// SIMATIC S7-200 project (STEP 7-Micro/WIN), CPU 224 CN REL 02.01

SYMBOL_TABLE 辅助
QDF              M1.0     // l运转启动
ZBF              M1.1     // 转速交变试验
WBF              M1.2     // 温度交变试验
GBF              M1.3     // 干温交变试验
ZBJSFW           M1.4     // 转速交变计数复位
WBJSFW           M1.5     // 温度交变计数复位
GBJSFW           M1.6     // 干湿交变计数复位
ZBWQ             M1.7     // 转速交变温控启动
WBWQ             M2.0     // 温度交变温控启动
GBWQ             M2.1     // 干温交变温控启动
                 M2.2     // 1号加热
                 M2.3     // 2号加热
                 M2.4     // 3号加热
                 M2.5     // 4号加热
                 M2.6     // 5号加热
                 M2.7     // 加热启动
F1               M3.0     // 1号气阀开
F2               M3.1     // 2号气阀开
F3               M3.2     // 3号气阀开
F4               M3.3     // 4号气阀开
F5               M3.4     // 5号气阀开
ZFF              M3.5     // 进口总气阀开
PF1              M3.6     // 室温自控
PF2              M3.7     // 强制排风
PF3              M4.0     // 排风辅助
FGDW             M4.1     // 阀门开到位
FKDW             M4.2     // 阀门关到位
F55              M4.3     // 5号气阀开
FXF              M4.4     // 皮带放松辅助
LJF              M4.5     // 皮带拉紧辅助
FXXWF            M4.6     // 放松限位辅助
LJXWF            M4.7     // 皮带限位辅助
DILJF            M5.0     // 手控拉紧辅助
DIFXF            M5.1     // 手控放松辅助
DILJFF           M5.2     // 手控拉紧辅助1
DIFXFF           M5.3     // 手控放松辅助1
HBF              M5.4     // 恒速试验
JS1F             M6.0     // 1号进水辅助
JS2F             M6.1     // 2号进水辅助
JS3F             M6.2     // 3号进水辅助
JS4F             M6.3     // 4号进水辅助
JS5F             M6.4     // 5号进水辅助
PS1F             M6.5     // 1号排水辅助
PS2F             M6.6     // 2号排水辅助
PS3F             M6.7     // 3号排水辅助
PS4F             M7.0     // 4号排水辅助
PS5F             M7.1     // 5号排水辅助
PSF              M7.2     // 排水辅助
JSF              M7.3     // 进水辅助
YWSF             M7.4     // 总水箱上限辅助
YWXF             M7.5     // 总水箱下限辅助
FZ1              M7.6     // 液位控制辅助1
FZ2              M7.7     // 液位控制辅助2
FZ3              M8.0     // 液位控制辅助3
FZ4              M8.1     // 液位控制辅助4
YWXF1            M8.2     // 液位下限辅助1
YWXF2            M8.3     // 液位下限辅助2
YWXF3            M8.4     // 液位下限辅助3
YWXF4            M8.5     // 液位下限辅助4
YWXF5            M8.6     // 液位下限辅助5
CYF              M8.7     // 采样辅助
WCF              M9.0     // 试验完成
SSJS             T101     // 转速上升时间
HSJS             T102     // 转速恒速时间
JSJS             T103     // 转速下降时间
GSSJS            T104     // 干湿交变加水时间
GSSJG            T105     // 干湿交变无水时间
                 T106     // 温度交变时间1
                 T107     // 温度交变时间2
                 T108     // 温度交变时间3
                 T109     // 温度交变时间4
                 T110     // 温度交变时间5
JR1SK            T111     // 1号箱加热控制时间
JR2SK            T112     // 2号箱加热控制时间
JR3SK            T113     // 3号箱加热控制时间
JR4SK            T114     // 4号箱加热控制时间
JR5SK            T115     // 5号箱加热控制时间
JRSZK            T116     // 加热间隔2秒延时
JRSZKF           T117     // 加热间隔2秒延时辅助
                 T46      // 采样时间
END_SYMBOL_TABLE

SYMBOL_TABLE 输入
                 I0.0     // 转速
FK               I0.1     // 电阀到位
YW1S             I0.2     // 1号箱水位上限
YW1X             I0.3     // 1号箱水位下限
YW2S             I0.4     // 2号箱水位上限
YW2X             I0.5     // 2号箱水位下限
YW3S             I0.6     // 3号箱水位上限
YW3X             I0.7     // 3号箱水位下限
YW4S             I1.0     // 4号箱水位上限
YW4X             I1.1     // 4号箱水位下限
YW5S             I1.2     // 5号箱水位上限
YW5X             I1.3     // 5号箱水位下限
YWS              I1.4     // 总箱水位上限
YWX              I1.5     // 总箱水位下限
FXW              I2.0     // 放松限位
LJW              I2.1     // 拉紧限位
DILJXC           I2.2     // 手控皮带拉紧
DIFXXC           I2.3     // 手控皮带放松
QD               I2.4     // 试验启动
TZ               I2.5     // 试验停止
DIDFK            I2.6     // 电阀开
DIDFG            I2.7     // 电阀关
DILJ             I3.0     // 手控皮带拉紧
DIFX             I3.1     // 手控皮带放松
DYQD             I3.2     // 电源启动
DYTZ             I3.3     // 电源停止
XL               I3.4     // 泄漏
CS               I3.5     // 水泵出水管有水
END_SYMBOL_TABLE

SYMBOL_TABLE 输出
DY               Q0.0     // 总电源
JRK              Q0.1     // 加热控制
JR1              Q0.2     // 加热1号箱
JR2              Q0.3     // 加热2号箱
JR3              Q0.4     // 加热3号箱
JR4              Q0.5     // 加热4号箱
JR5              Q0.6     // 加热5号箱
DFK              Q0.7     // 电阀开
DFG              Q1.0     // 电阀关
LJ               Q1.1     // 电机拉紧
FX               Q2.0     // 电机放松
PF               Q2.1     // 排风扇
ZYF              Q2.2     // 增压阀F18
PYF              Q2.3     // 排空阀F19
QF1              Q2.4     // 1号箱气阀F12
QF2              Q2.5     // 2号箱气阀F13
QF3              Q2.6     // 3号箱气阀F14
QF4              Q2.7     // 4号箱气阀F15
QF5              Q3.0     // 5号箱气阀F16
ZQF              Q3.1     // 总控气阀FF17
JS1              Q3.2     // 1号箱进水F3
JS2              Q3.3     // 2号箱进水F4
JS3              Q3.4     // 3号箱进水F5
JS4              Q3.5     // 4号箱进水F6
JS5              Q3.6     // 5号箱进水F7
ZJS              Q3.7     // 总进水F1
ZPS              Q4.0     // 总排水F2
ZKF              Q4.1     // 总水箱控制F8
CKJQF            Q4.2     // 水泵出水管进气F11
JKPSF            Q4.3     // 水泵进水管排水F9
ZSXJY            Q4.4     // 总水箱加压(水盆回水)F10
NZ               Q4.5     // 逆转
SZ               Q4.6     // 顺转
END_SYMBOL_TABLE

SYMBOL_TABLE 变量
XTQD             VB201    // ＝0停止　＝1启动
ZDFX             VB202    // 转动方向＝0顺时运转　＝0逆时运转
SYLX             VB203    // 系统停止＝0　转速交变＝1　温度交变＝2　干交变＝3
PKQD             VB204    // 压力控制=0停止=1自动
YZZT             VB205    // 运转状态＝0停止＝1升速　＝2恒速　＝3降速
WKQD             VB206    // =0加热停止 =1加热启动
HKZ              VB207    // 扬程控制=0手控 =1自控
YWKZ             VB208    // 液位控制=0手控 =1自控
WBSL             VB209    // 温变数量
WBBK             VB210    // 温变步控
LLKZ             VB211    // 拉力控制=0停止=1自动
SBZT             VB212    // 试验状态=0正常 =1 泄漏 =2结束
XLCY             VB214    // 允许泄漏报警
ZPC              VD150    // 转速交变频次
WPC              VD154    // 温度交变频次
GPC              VD158    // 干湿交变频次
H                VW100    // 扬程
P                VW102    // 水箱压力
LL               VW104    // 皮带拉力
WD1              VW106    // 水温1
WD2              VW108    // 水温2
WD3              VW110    // 水温3
WD4              VW112    // 水温4
WD5              VW114    // 水温5
SW               VW116    // 室温
N                VW118    // 转速
FW               VW120    // 阀位
LLSD             VW122    // 拉力设定
PSD              VW124    // 压力设定
HSD              VW126    // 扬程设定
ZSJ              VW128    // 状态运行时间
WD1SD            VW130    // 温度设定1
WD2SD            VW132    // 温度设定2
WD3SD            VW134    // 温度设定3
WD4SD            VW136    // 温度设定4
WD5SD            VW138    // 温度设定5
SJSD1            VW140    // 时间设定1
SJSD2            VW142    // 时间设定2
SJSD3            VW144    // 时间设定3
SJSD4            VW146    // 时间设定4
SJSD5            VW148    // 时间设定5
WD1WC            VW306    // 1号箱温差
WD2WC            VW308    // 2号箱温差
WD3WC            VW310    // 3号箱温差
WD4WC            VW312    // 4号箱温差
WD5WC            VW314    // 5号箱温差
HMAX             VW316    // 扬程上限N
HMIN             VW318    // 扬程下限N
LLMAX            VW320    // 拉力上限N
LLMIN            VW322    // 拉力下限N
PMAX             VW356    // 压力上限
PMIN             VW358    // 压力下限
WD1WCF           VW378    // 1号箱温度差
WD2WCF           VW380    // 2号箱温度差
WD3WCF           VW382    // 3号箱温度差
WD4WCF           VW384    // 4号箱温度差
WD5WCF           VW386    // 5号箱温度差
END_SYMBOL_TABLE

ORGANIZATION_BLOCK 程序块:OB1
TITLE=程序注释
BEGIN
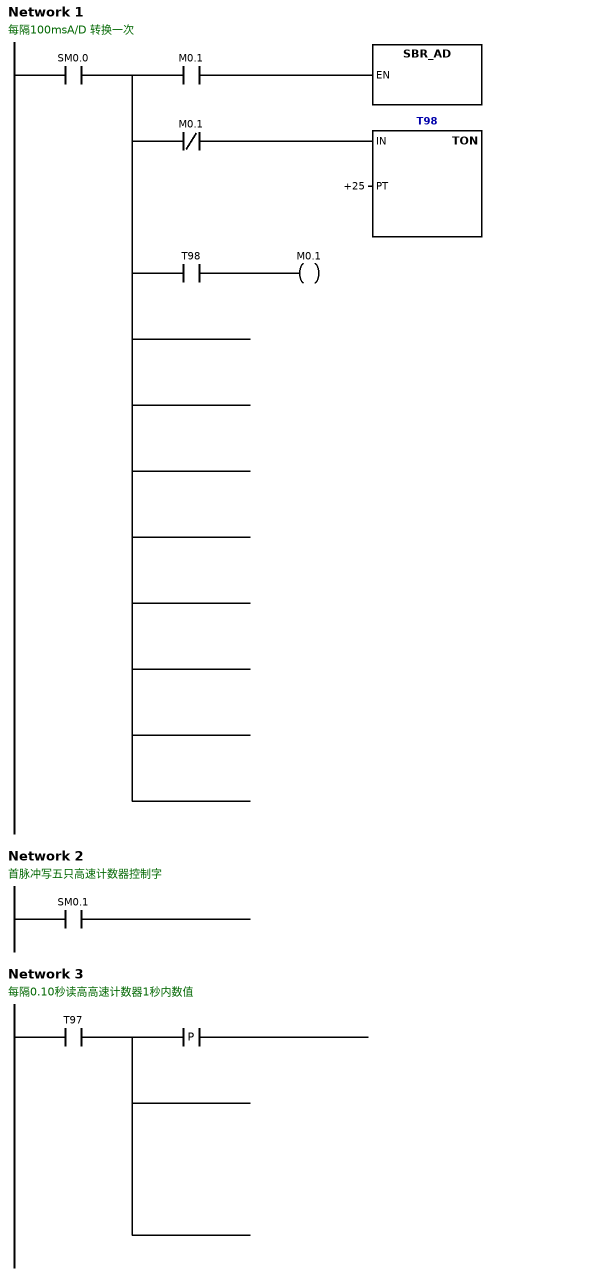
Network 1
// 每隔100msA/D 转换一次
// (network saved uncompiled; LAD cells follow)
// row 0: c0 -| |- SM0.0 v  c1 -| |- M0.1  c2 --  c3 [SBR_AD EN:=power@row0]
// row 1: c0 ^v  c1 -|/|- M0.1  c2 --  c3 [TON T98 IN:=power@row1, PT:=+25]
// row 2: c0 ^v  c3 [box]
// row 3: c0 ^v  c1 -| |- T98  c2 -( ) M0.1
// row 4: c0 ^v  c1 --
// row 5: c0 ^v  c1 --
// row 6: c0 ^v  c1 --
// row 7: c0 ^v  c1 --
// row 8: c0 ^v  c1 --
// row 9: c0 ^v  c1 --
// row 10: c0 ^v  c1 --
// row 11: c0 ^  c1 --
Network 2
// 首脉冲写五只高速计数器控制字
// (network saved uncompiled; LAD cells follow)
// row 0: c0 -| |- SM0.1  c1 --
Network 3
// 每隔0.10秒读高高速计数器1秒内数值
// (network saved uncompiled; LAD cells follow)
// row 0: c0 -| |- T97 v  c1 -|P|-  c2 --
// row 1: c0 ^v  c1 --
// row 2: c0 ^v
// row 3: c0 ^  c1 --
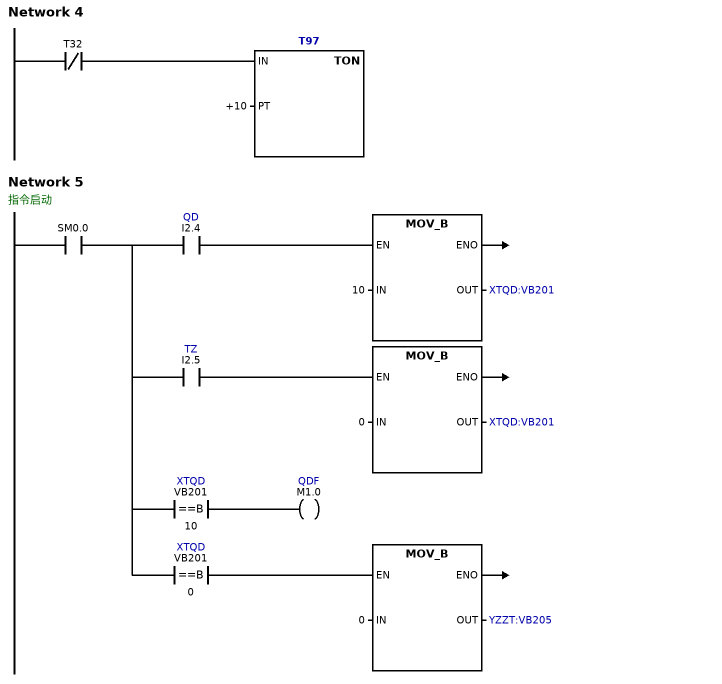
Network 4
LDN    T32
TON    T97, +10
Network 5
// 指令启动
LD     SM0.0
LPS
A      QD:I2.4
MOVB   10, XTQD:VB201
LRD
A      TZ:I2.5
MOVB   0, XTQD:VB201
LRD
AB=    XTQD:VB201, 10
=      QDF:M1.0
LPP
AB=    XTQD:VB201, 0
MOVB   0, YZZT:VB205
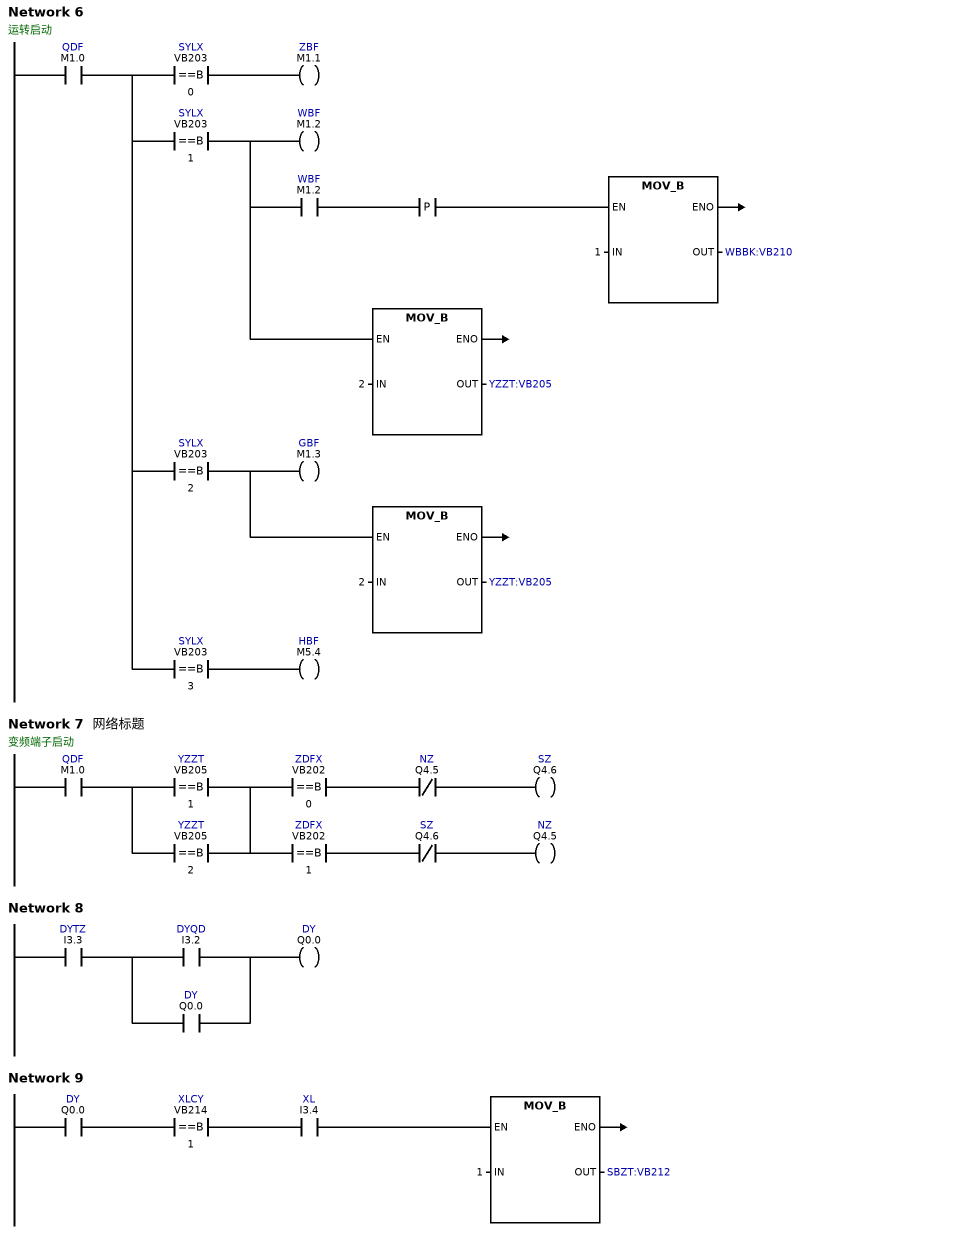
Network 6
// 运转启动
LD     QDF:M1.0
LPS
AB=    SYLX:VB203, 0
=      ZBF:M1.1
LRD
AB=    SYLX:VB203, 1
LPS
=      WBF:M1.2
A      WBF:M1.2
EU
MOVB   1, WBBK:VB210
LPP
MOVB   2, YZZT:VB205
LRD
AB=    SYLX:VB203, 2
=      GBF:M1.3
MOVB   2, YZZT:VB205
LPP
AB=    SYLX:VB203, 3
=      HBF:M5.4
Network 7 // 网络标题
// 变频端子启动
LD     QDF:M1.0
LDB=   YZZT:VB205, 1
OB=    YZZT:VB205, 2
ALD
LPS
AB=    ZDFX:VB202, 0
AN     NZ:Q4.5
=      SZ:Q4.6
LPP
AB=    ZDFX:VB202, 1
AN     SZ:Q4.6
=      NZ:Q4.5
Network 8
LD     DYTZ:I3.3
LD     DYQD:I3.2
O      DY:Q0.0
ALD
=      DY:Q0.0
Network 9
LD     DY:Q0.0
AB=    XLCY:VB214, 1
A      XL:I3.4
MOVB   1, SBZT:VB212
Network 18 // 网络标题
// 网络注释
END_ORGANIZATION_BLOCK

SUBROUTINE_BLOCK SBR_AD:SBR0
TITLE=子例行程序注释
BEGIN
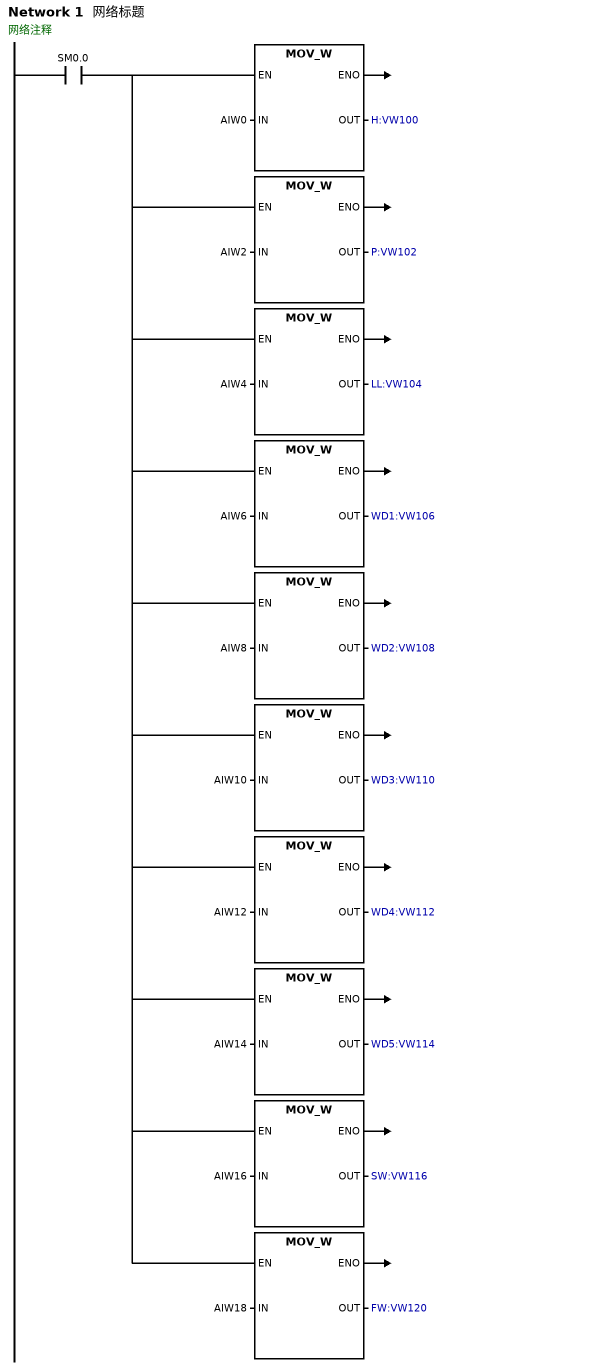
Network 1 // 网络标题
// 网络注释
LD     SM0.0
MOVW   AIW0, H:VW100
MOVW   AIW2, P:VW102
MOVW   AIW4, LL:VW104
MOVW   AIW6, WD1:VW106
MOVW   AIW8, WD2:VW108
MOVW   AIW10, WD3:VW110
MOVW   AIW12, WD4:VW112
MOVW   AIW14, WD5:VW114
MOVW   AIW16, SW:VW116
MOVW   AIW18, FW:VW120
Network 11 // 网络标题
// 网络注释
END_SUBROUTINE_BLOCK

SUBROUTINE_BLOCK 干湿交变:SBR1
TITLE=子例行程序注释
BEGIN
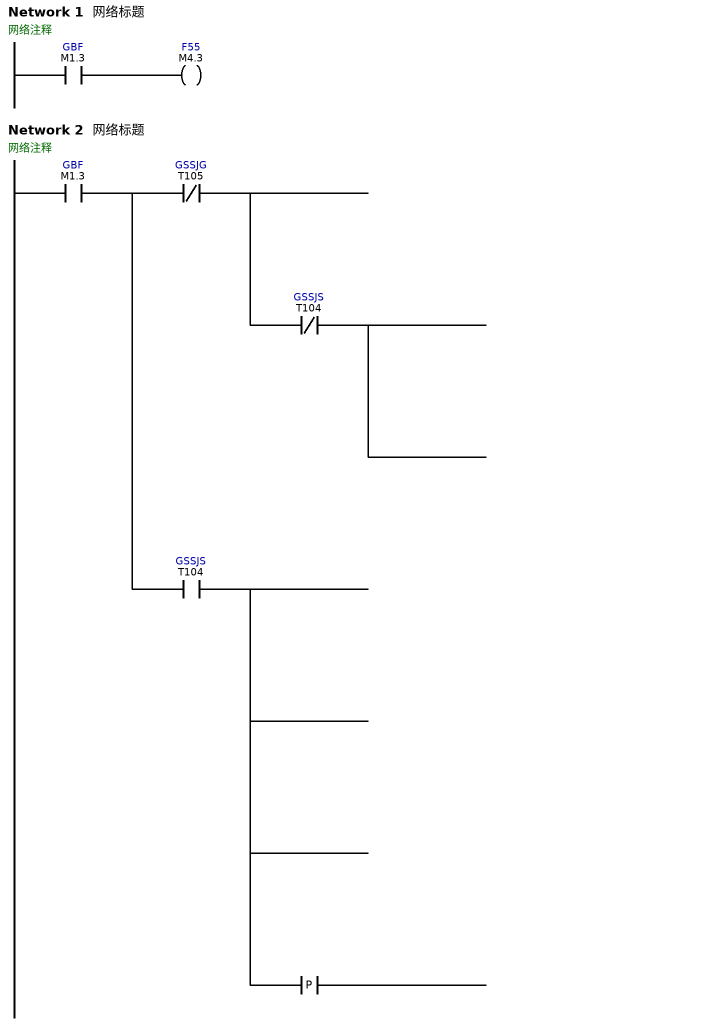
Network 1 // 网络标题
// 网络注释
LD     GBF:M1.3
=      F55:M4.3
Network 2 // 网络标题
// 网络注释
// (network saved uncompiled; LAD cells follow)
// row 0: c0 -| |- GBF:M1.3 v  c1 -|/|- GSSJG:T105 v  c2 --
// row 1: c0 ^v  c1 ^v
// row 2: c0 ^v  c1 ^  c2 -|/|- GSSJS:T104 v  c3 --
// row 3: c0 ^v  c2 ^v
// row 4: c0 ^v  c2 ^  c3 --
// row 5: c0 ^v
// row 6: c0 ^  c1 -| |- GSSJS:T104 v  c2 --
// row 7: c1 ^v
// row 8: c1 ^v  c2 --
// row 9: c1 ^v
// row 10: c1 ^v  c2 --
// row 11: c1 ^v
// row 12: c1 ^  c2 -|P|-  c3 --
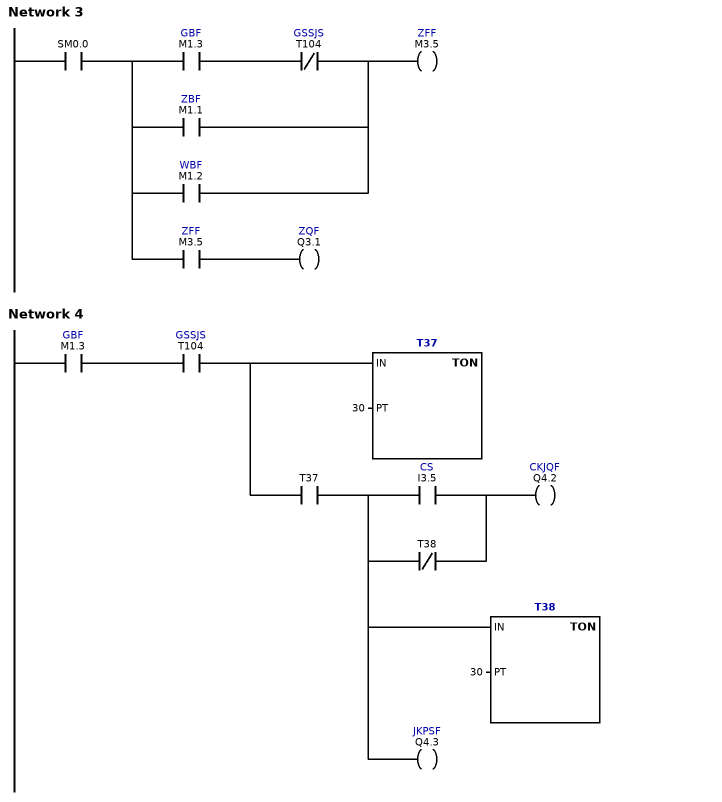
Network 3
LD     SM0.0
LPS
LD     GBF:M1.3
AN     GSSJS:T104
O      ZBF:M1.1
O      WBF:M1.2
ALD
=      ZFF:M3.5
LPP
A      ZFF:M3.5
=      ZQF:Q3.1
Network 4
LD     GBF:M1.3
A      GSSJS:T104
TON    T37, 30
A      T37
LPS
LD     CS:I3.5
ON     T38
ALD
=      CKJQF:Q4.2
LPP
TON    T38, 30
=      JKPSF:Q4.3
END_SUBROUTINE_BLOCK

SUBROUTINE_BLOCK 水温控制:SBR2
TITLE=子例行程序注释
BEGIN
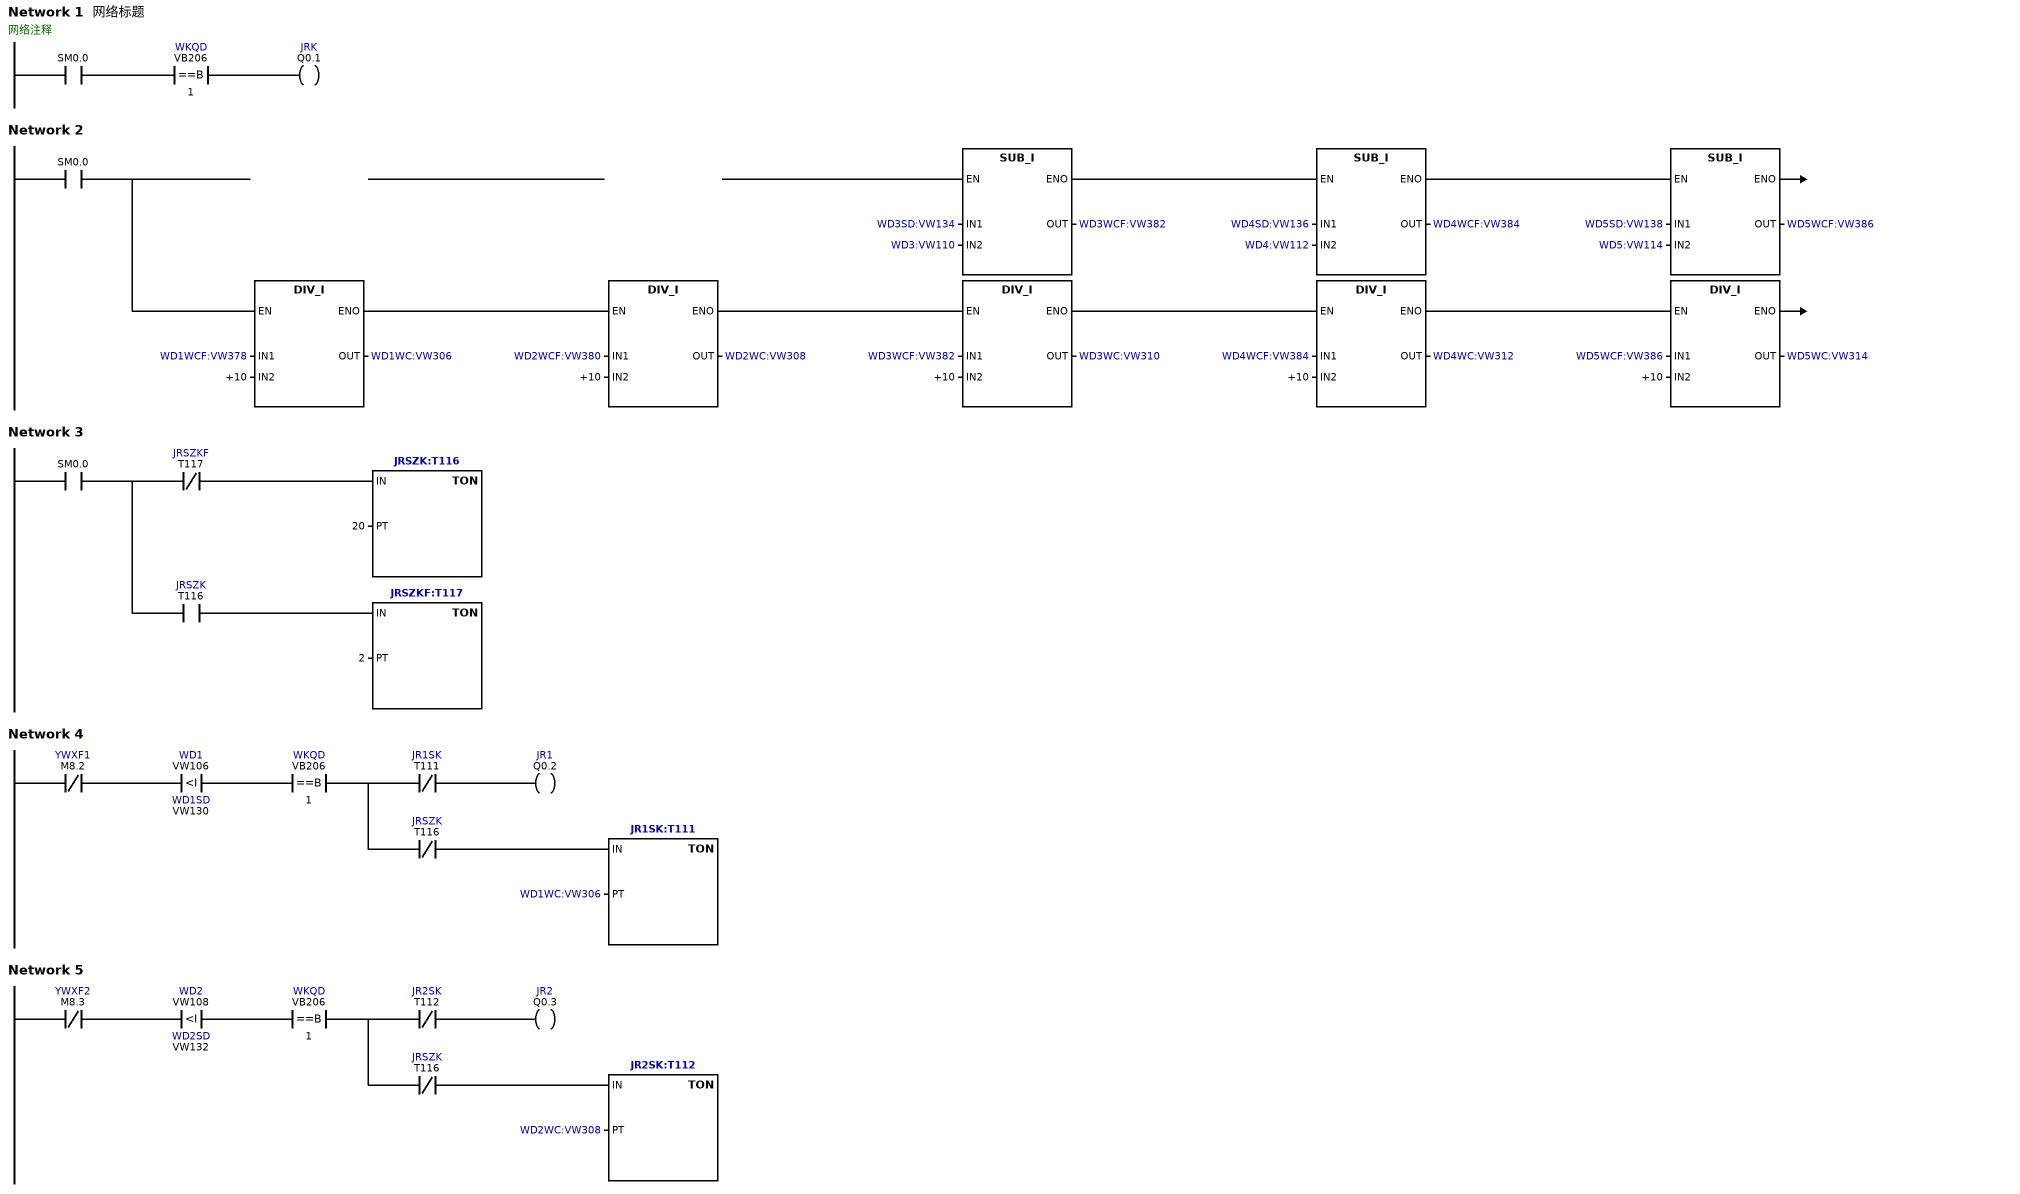
Network 1 // 网络标题
// 网络注释
LD     SM0.0
AB=    WKQD:VB206, 1
=      JRK:Q0.1
Network 2
// (network saved uncompiled; LAD cells follow)
// row 0: c0 -| |- SM0.0 v  c1 --  c3 --  c4 --  c6 --  c7 --  c8 [SUB_I EN:=power@row0, IN1:=WD3SD:VW134, IN2:=WD3:VW110, ENO=>power, OUT=>WD3WCF:VW382]  c9 --  c10 --  c11 [SUB_I EN:=power@row0, IN1:=WD4SD:VW136, IN2:=WD4:VW112, ENO=>power, OUT=>WD4WCF:VW384]  c12 --  c13 --  c14 [SUB_I EN:=power@row0, IN1:=WD5SD:VW138, IN2:=WD5:VW114, ENO=>power, OUT=>WD5WCF:VW386]  c15 ->
// row 1: c0 ^v  c8 [box]  c11 [box]  c14 [box]
// row 2: c0 ^  c1 --  c2 [DIV_I EN:=power@row2, IN1:=WD1WCF:VW378, IN2:=+10, ENO=>power, OUT=>WD1WC:VW306]  c3 --  c4 --  c5 [DIV_I EN:=power@row2, IN1:=WD2WCF:VW380, IN2:=+10, ENO=>power, OUT=>WD2WC:VW308]  c6 --  c7 --  c8 [DIV_I EN:=power@row2, IN1:=WD3WCF:VW382, IN2:=+10, ENO=>power, OUT=>WD3WC:VW310]  c9 --  c10 --  c11 [DIV_I EN:=power@row2, IN1:=WD4WCF:VW384, IN2:=+10, ENO=>power, OUT=>WD4WC:VW312]  c12 --  c13 --  c14 [DIV_I EN:=power@row2, IN1:=WD5WCF:VW386, IN2:=+10, ENO=>power, OUT=>WD5WC:VW314]  c15 ->
// row 3: c2 [box]  c5 [box]  c8 [box]  c11 [box]  c14 [box]
Network 3
LD     SM0.0
LPS
AN     JRSZKF:T117
TON    JRSZK:T116, 20
LPP
A      JRSZK:T116
TON    JRSZKF:T117, 2
Network 4
LDN    YWXF1:M8.2
AW<    WD1:VW106, WD1SD:VW130
AB=    WKQD:VB206, 1
LPS
AN     JR1SK:T111
=      JR1:Q0.2
LPP
AN     JRSZK:T116
TON    JR1SK:T111, WD1WC:VW306
Network 5
LDN    YWXF2:M8.3
AW<    WD2:VW108, WD2SD:VW132
AB=    WKQD:VB206, 1
LPS
AN     JR2SK:T112
=      JR2:Q0.3
LPP
AN     JRSZK:T116
TON    JR2SK:T112, WD2WC:VW308
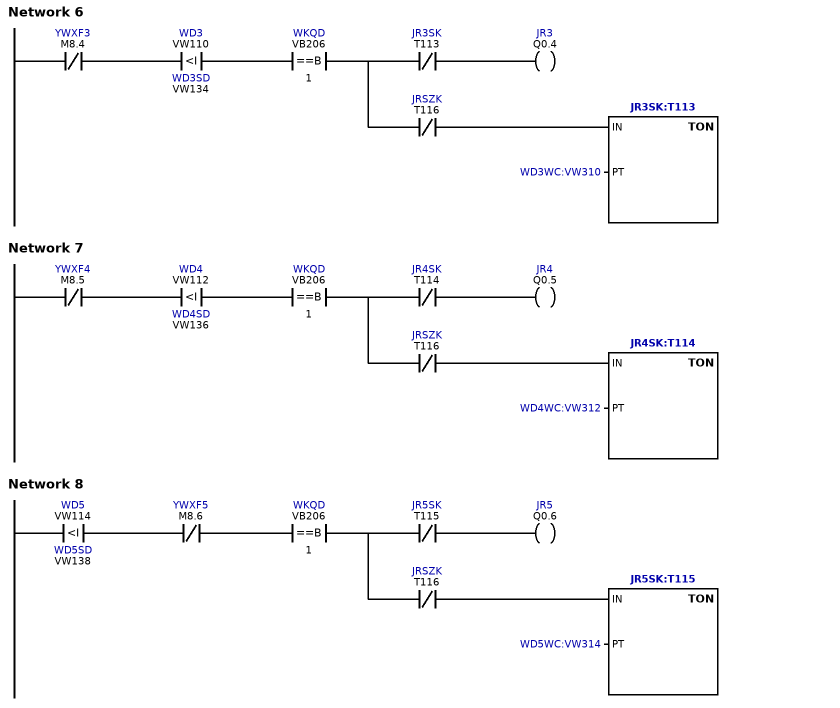
Network 6
LDN    YWXF3:M8.4
AW<    WD3:VW110, WD3SD:VW134
AB=    WKQD:VB206, 1
LPS
AN     JR3SK:T113
=      JR3:Q0.4
LPP
AN     JRSZK:T116
TON    JR3SK:T113, WD3WC:VW310
Network 7
LDN    YWXF4:M8.5
AW<    WD4:VW112, WD4SD:VW136
AB=    WKQD:VB206, 1
LPS
AN     JR4SK:T114
=      JR4:Q0.5
LPP
AN     JRSZK:T116
TON    JR4SK:T114, WD4WC:VW312
Network 8
LDW<   WD5:VW114, WD5SD:VW138
AN     YWXF5:M8.6
AB=    WKQD:VB206, 1
LPS
AN     JR5SK:T115
=      JR5:Q0.6
LPP
AN     JRSZK:T116
TON    JR5SK:T115, WD5WC:VW314
END_SUBROUTINE_BLOCK

SUBROUTINE_BLOCK 皮带拉力:SBR4
TITLE=子例行程序注释
BEGIN
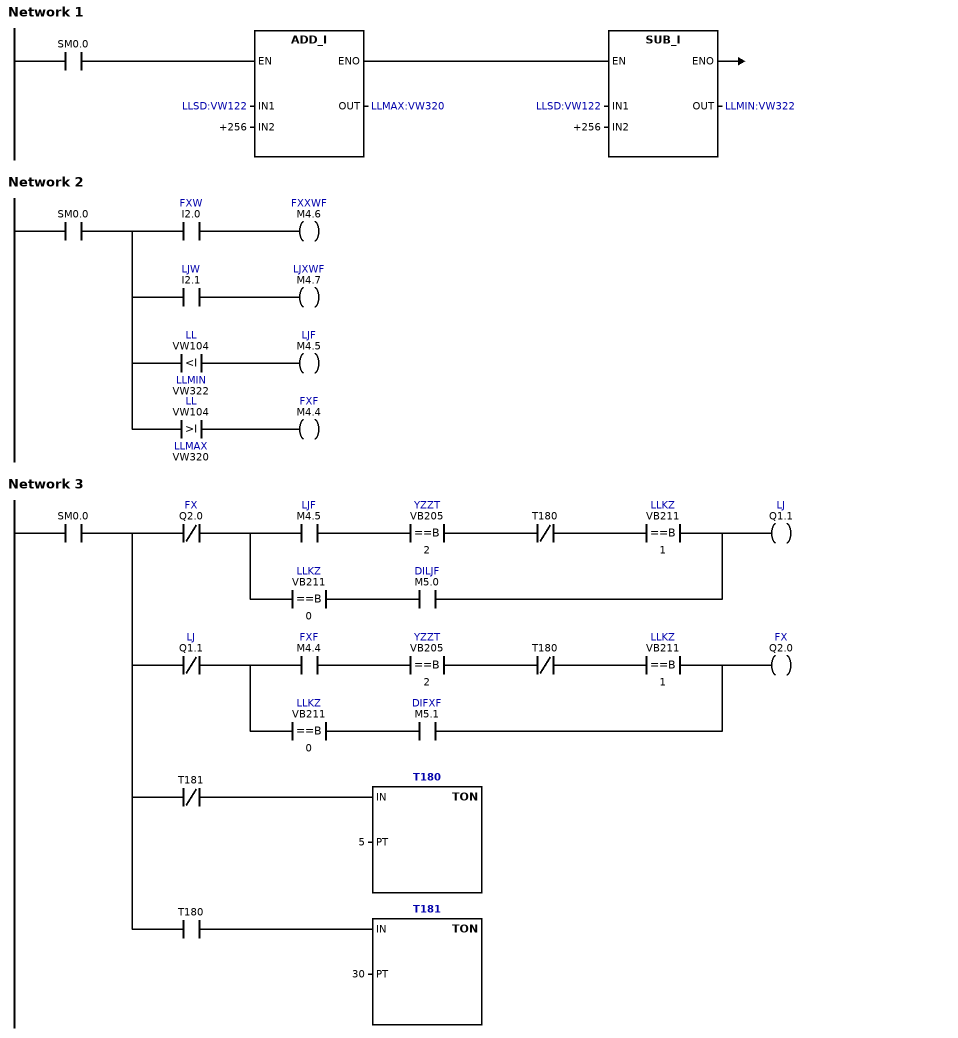
Network 1
LD     SM0.0
MOVW   LLSD:VW122, LLMAX:VW320
AENO
+I     +256, LLMAX:VW320
AENO
MOVW   LLSD:VW122, LLMIN:VW322
-I     +256, LLMIN:VW322
Network 2
LD     SM0.0
LPS
A      FXW:I2.0
=      FXXWF:M4.6
LRD
A      LJW:I2.1
=      LJXWF:M4.7
LRD
AW<    LL:VW104, LLMIN:VW322
=      LJF:M4.5
LPP
AW>    LL:VW104, LLMAX:VW320
=      FXF:M4.4
Network 3
LD     SM0.0
LPS
AN     FX:Q2.0
LD     LJF:M4.5
AB=    YZZT:VB205, 2
AN     T180
AB=    LLKZ:VB211, 1
LDB=   LLKZ:VB211, 0
A      DILJF:M5.0
OLD
ALD
=      LJ:Q1.1
LRD
AN     LJ:Q1.1
LD     FXF:M4.4
AB=    YZZT:VB205, 2
AN     T180
AB=    LLKZ:VB211, 1
LDB=   LLKZ:VB211, 0
A      DIFXF:M5.1
OLD
ALD
=      FX:Q2.0
LPP
LPS
AN     T181
TON    T180, 5
LPP
A      T180
TON    T181, 30
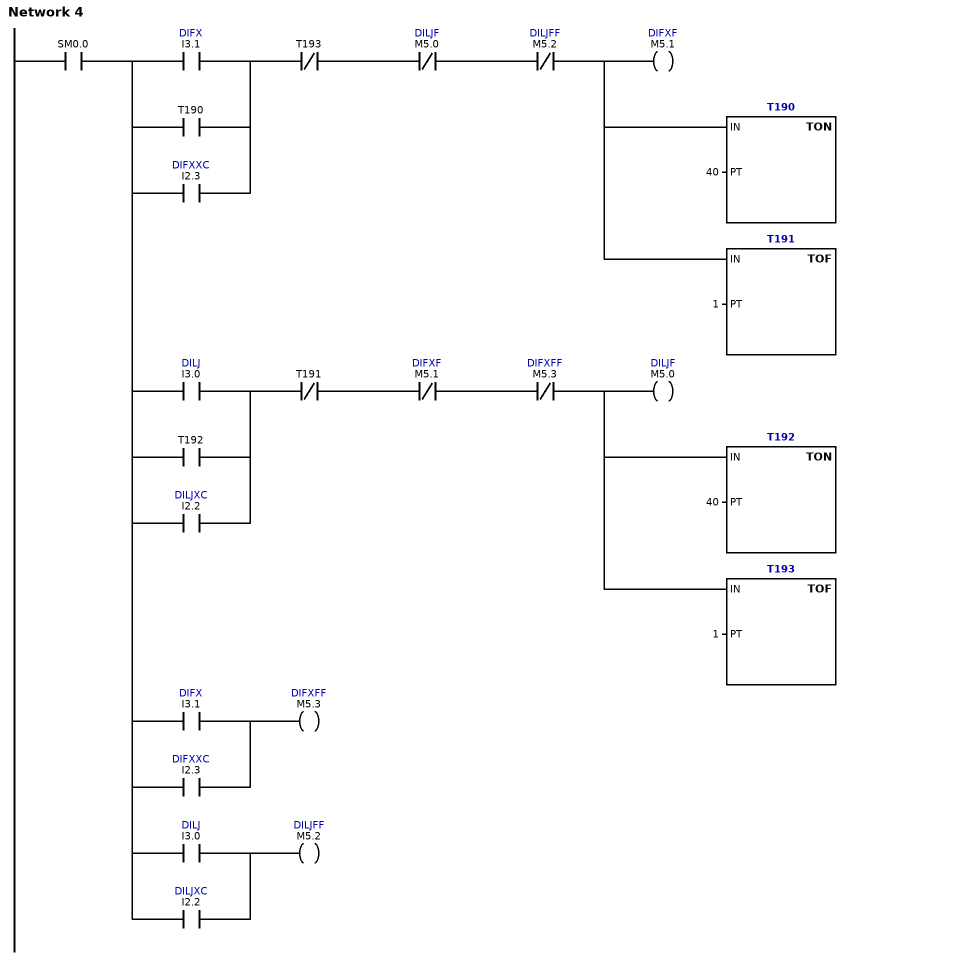
Network 4
LD     SM0.0
LPS
LD     DIFX:I3.1
O      T190
O      DIFXXC:I2.3
AN     T193
AN     DILJF:M5.0
AN     DILJFF:M5.2
ALD
=      DIFXF:M5.1
TON    T190, 40
TOF    T191, 1
LRD
LD     DILJ:I3.0
O      T192
O      DILJXC:I2.2
AN     T191
AN     DIFXF:M5.1
AN     DIFXFF:M5.3
ALD
=      DILJF:M5.0
TON    T192, 40
TOF    T193, 1
LRD
LD     DIFX:I3.1
O      DIFXXC:I2.3
ALD
=      DIFXFF:M5.3
LPP
LD     DILJ:I3.0
O      DILJXC:I2.2
ALD
=      DILJFF:M5.2
END_SUBROUTINE_BLOCK

SUBROUTINE_BLOCK HSC_清零:SBR5
TITLE=子例行程序注释
BEGIN
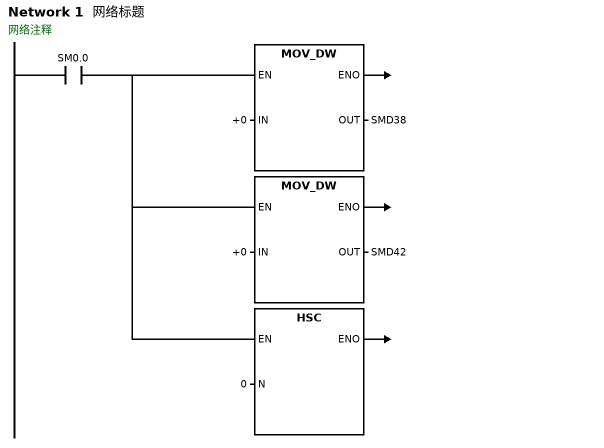
Network 1 // 网络标题
// 网络注释
LD     SM0.0
MOVD   +0, SMD38
MOVD   +0, SMD42
HSC    0
END_SUBROUTINE_BLOCK

SUBROUTINE_BLOCK 温度交变:SBR6
TITLE=子例行程序注释
BEGIN
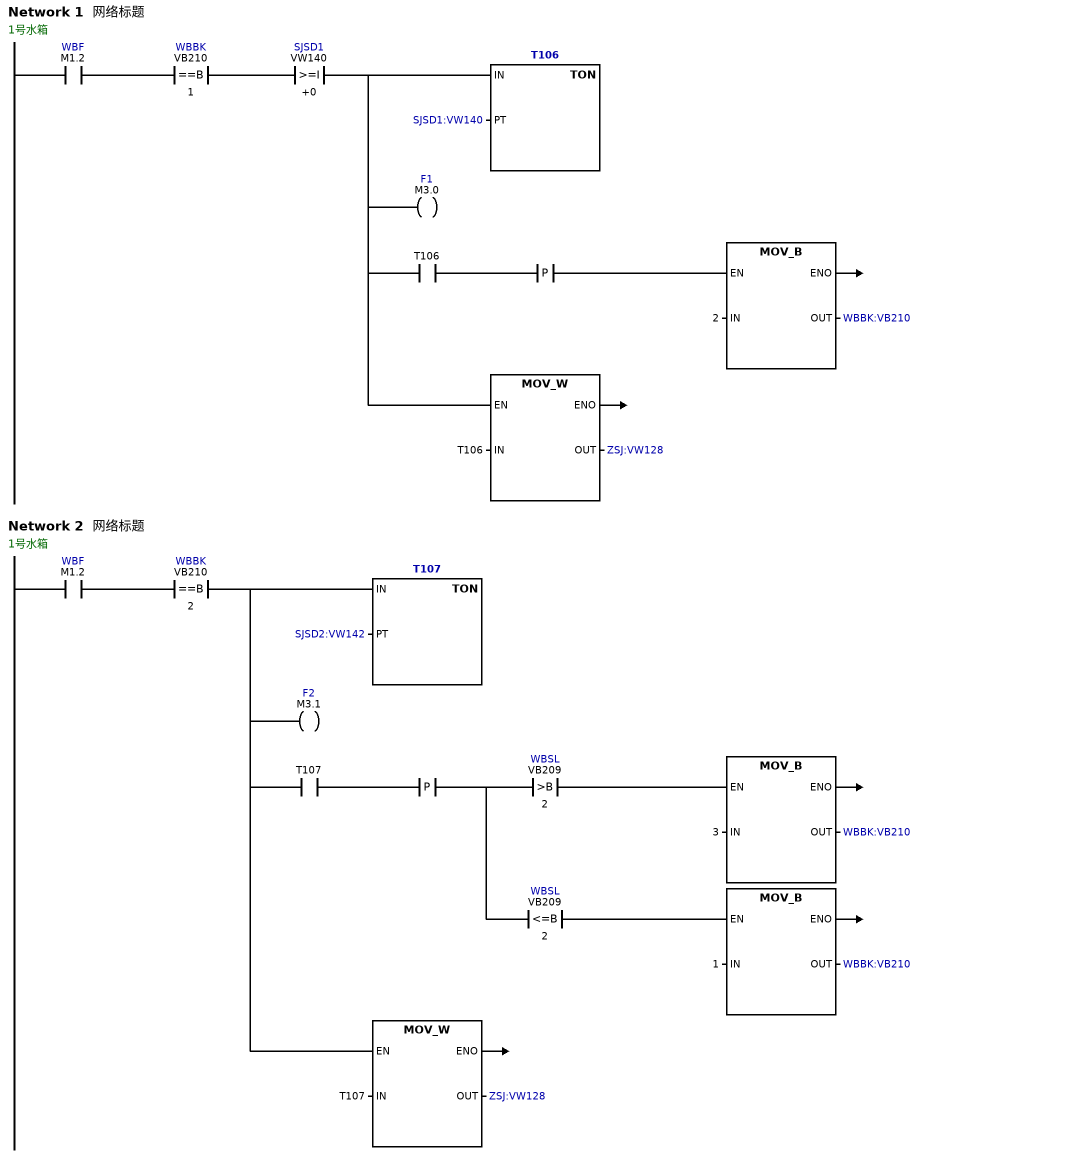
Network 1 // 网络标题
// 1号水箱
LD     WBF:M1.2
AB=    WBBK:VB210, 1
AW>=   SJSD1:VW140, +0
LPS
TON    T106, SJSD1:VW140
=      F1:M3.0
A      T106
EU
MOVB   2, WBBK:VB210
LPP
MOVW   T106, ZSJ:VW128
Network 2 // 网络标题
// 1号水箱
LD     WBF:M1.2
AB=    WBBK:VB210, 2
LPS
TON    T107, SJSD2:VW142
=      F2:M3.1
A      T107
EU
LPS
AB>    WBSL:VB209, 2
MOVB   3, WBBK:VB210
LPP
AB<=   WBSL:VB209, 2
MOVB   1, WBBK:VB210
LPP
MOVW   T107, ZSJ:VW128
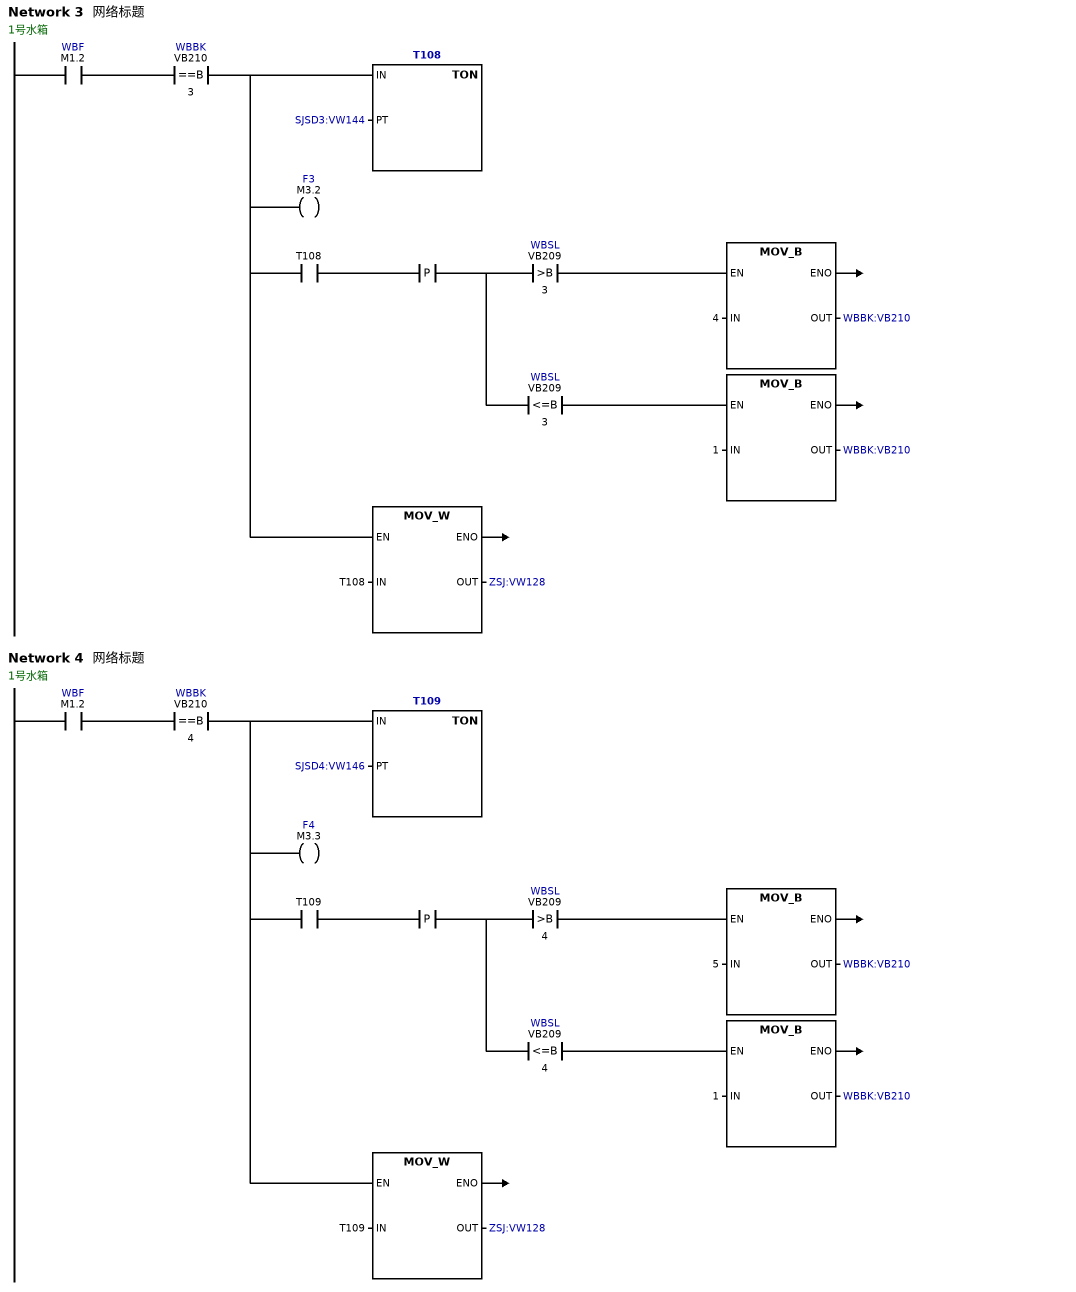
Network 3 // 网络标题
// 1号水箱
LD     WBF:M1.2
AB=    WBBK:VB210, 3
LPS
TON    T108, SJSD3:VW144
=      F3:M3.2
A      T108
EU
LPS
AB>    WBSL:VB209, 3
MOVB   4, WBBK:VB210
LPP
AB<=   WBSL:VB209, 3
MOVB   1, WBBK:VB210
LPP
MOVW   T108, ZSJ:VW128
Network 4 // 网络标题
// 1号水箱
LD     WBF:M1.2
AB=    WBBK:VB210, 4
LPS
TON    T109, SJSD4:VW146
=      F4:M3.3
A      T109
EU
LPS
AB>    WBSL:VB209, 4
MOVB   5, WBBK:VB210
LPP
AB<=   WBSL:VB209, 4
MOVB   1, WBBK:VB210
LPP
MOVW   T109, ZSJ:VW128
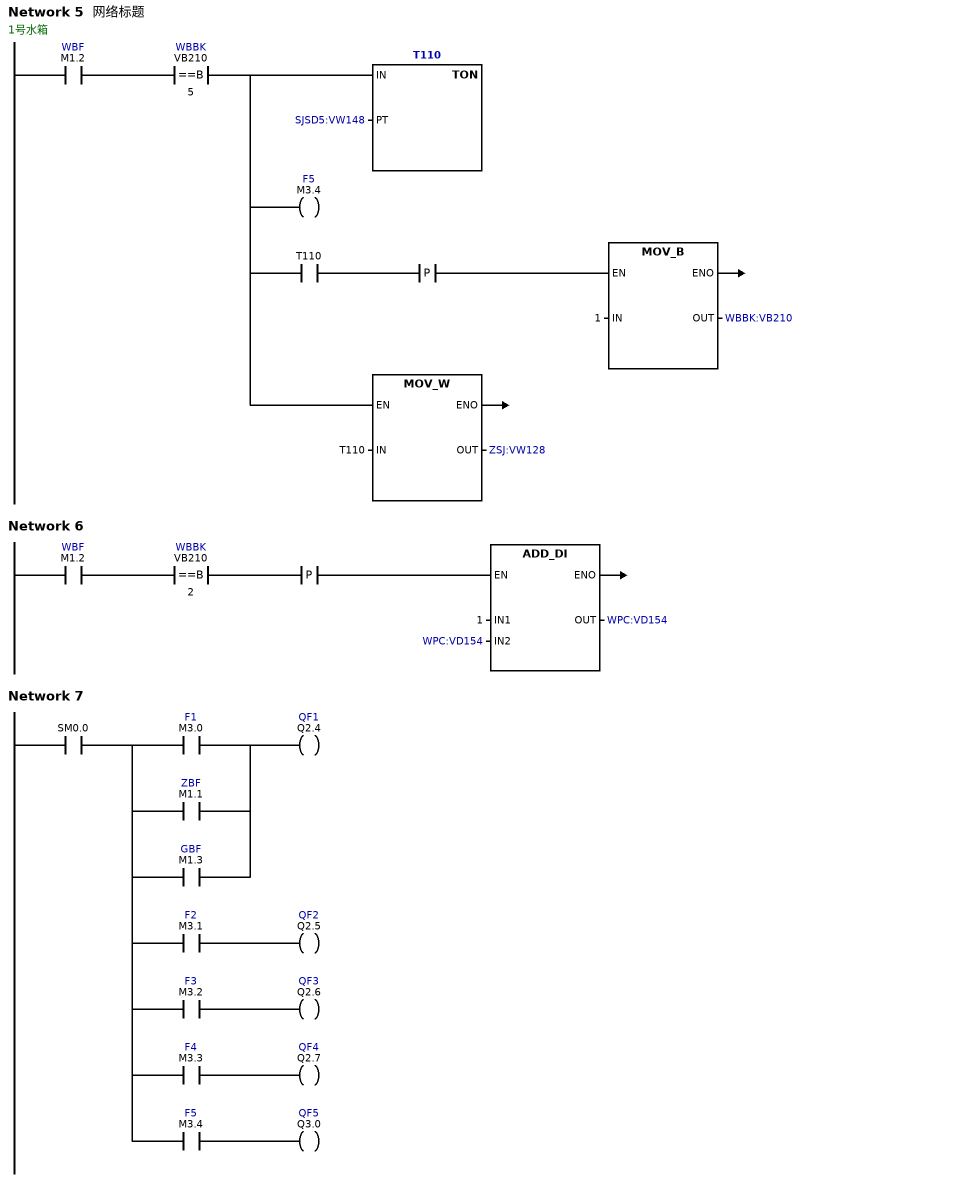
Network 5 // 网络标题
// 1号水箱
LD     WBF:M1.2
AB=    WBBK:VB210, 5
LPS
TON    T110, SJSD5:VW148
=      F5:M3.4
A      T110
EU
MOVB   1, WBBK:VB210
LPP
MOVW   T110, ZSJ:VW128
Network 6
LD     WBF:M1.2
AB=    WBBK:VB210, 2
EU
+D     1, WPC:VD154
Network 7
LD     SM0.0
LPS
LD     F1:M3.0
O      ZBF:M1.1
O      GBF:M1.3
ALD
=      QF1:Q2.4
LPP
LPS
A      F2:M3.1
=      QF2:Q2.5
LRD
A      F3:M3.2
=      QF3:Q2.6
LRD
A      F4:M3.3
=      QF4:Q2.7
LPP
A      F5:M3.4
=      QF5:Q3.0
END_SUBROUTINE_BLOCK

SUBROUTINE_BLOCK 液位控制:SBR7
TITLE=子程序注释
BEGIN
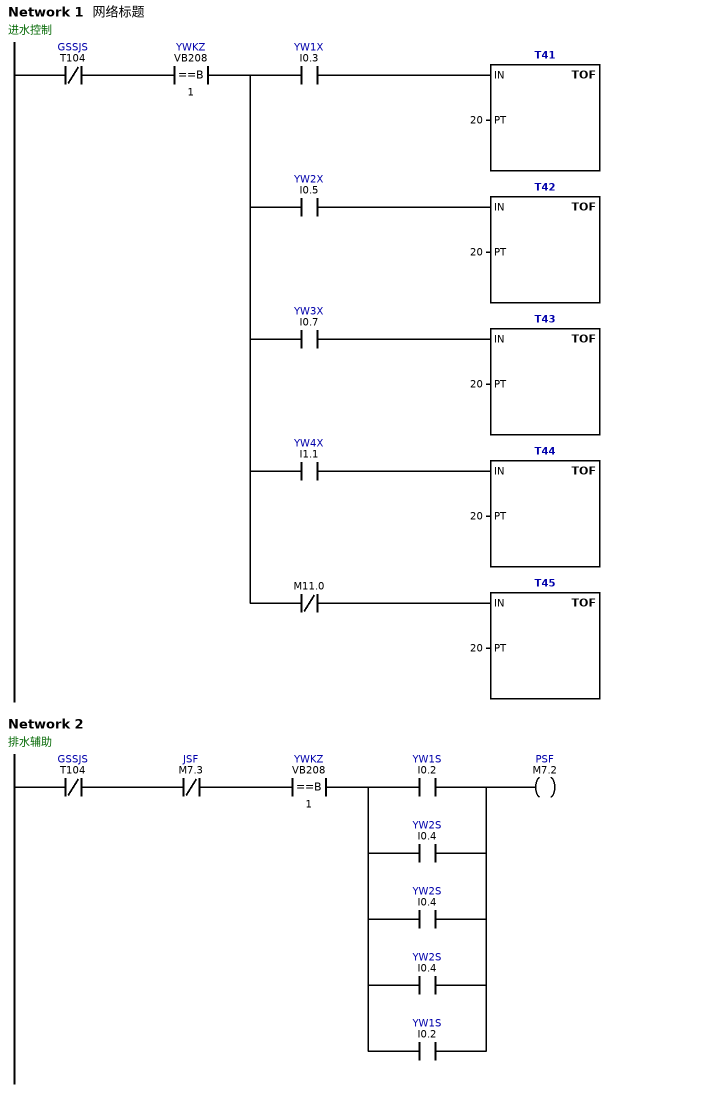
Network 1 // 网络标题
// 进水控制
LDN    GSSJS:T104
AB=    YWKZ:VB208, 1
LPS
A      YW1X:I0.3
TOF    T41, 20
LRD
A      YW2X:I0.5
TOF    T42, 20
LRD
A      YW3X:I0.7
TOF    T43, 20
LRD
A      YW4X:I1.1
TOF    T44, 20
LPP
AN     M11.0
TOF    T45, 20
Network 2
// 排水辅助
LDN    GSSJS:T104
AN     JSF:M7.3
AB=    YWKZ:VB208, 1
LD     YW1S:I0.2
O      YW2S:I0.4
O      YW2S:I0.4
O      YW2S:I0.4
O      YW1S:I0.2
ALD
=      PSF:M7.2
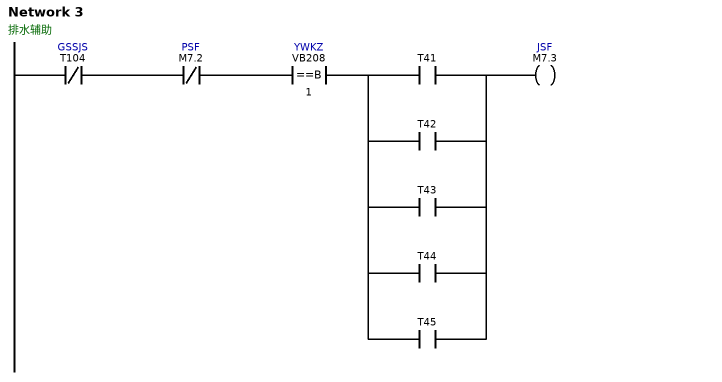
Network 3
// 排水辅助
LDN    GSSJS:T104
AN     PSF:M7.2
AB=    YWKZ:VB208, 1
LD     T41
O      T42
O      T43
O      T44
O      T45
ALD
=      JSF:M7.3
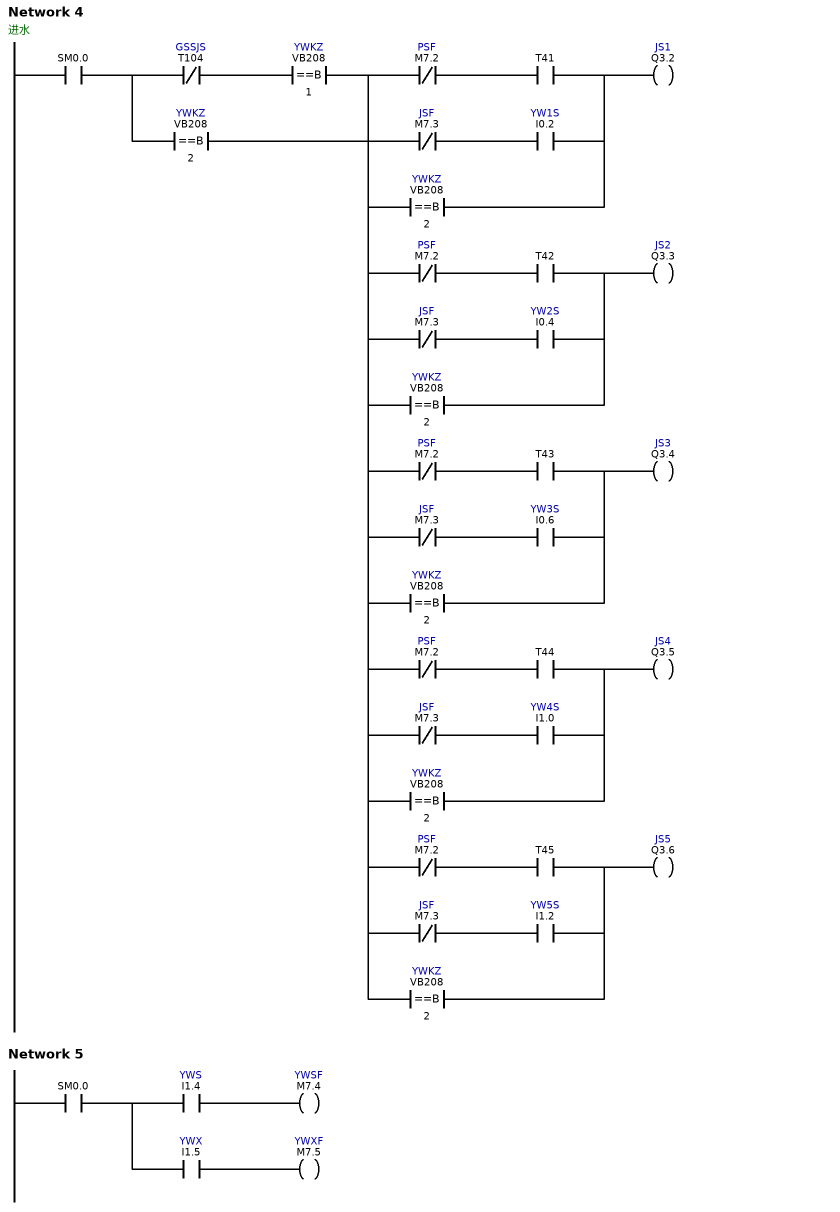
Network 4
// 进水
LD     SM0.0
LDN    GSSJS:T104
AB=    YWKZ:VB208, 1
OB=    YWKZ:VB208, 2
ALD
LPS
LDN    PSF:M7.2
A      T41
LDN    JSF:M7.3
A      YW1S:I0.2
OLD
OB=    YWKZ:VB208, 2
ALD
=      JS1:Q3.2
LRD
LDN    PSF:M7.2
A      T42
LDN    JSF:M7.3
A      YW2S:I0.4
OLD
OB=    YWKZ:VB208, 2
ALD
=      JS2:Q3.3
LRD
LDN    PSF:M7.2
A      T43
LDN    JSF:M7.3
A      YW3S:I0.6
OLD
OB=    YWKZ:VB208, 2
ALD
=      JS3:Q3.4
LRD
LDN    PSF:M7.2
A      T44
LDN    JSF:M7.3
A      YW4S:I1.0
OLD
OB=    YWKZ:VB208, 2
ALD
=      JS4:Q3.5
LPP
LDN    PSF:M7.2
A      T45
LDN    JSF:M7.3
A      YW5S:I1.2
OLD
OB=    YWKZ:VB208, 2
ALD
=      JS5:Q3.6
Network 5
LD     SM0.0
LPS
A      YWS:I1.4
=      YWSF:M7.4
LPP
A      YWX:I1.5
=      YWXF:M7.5
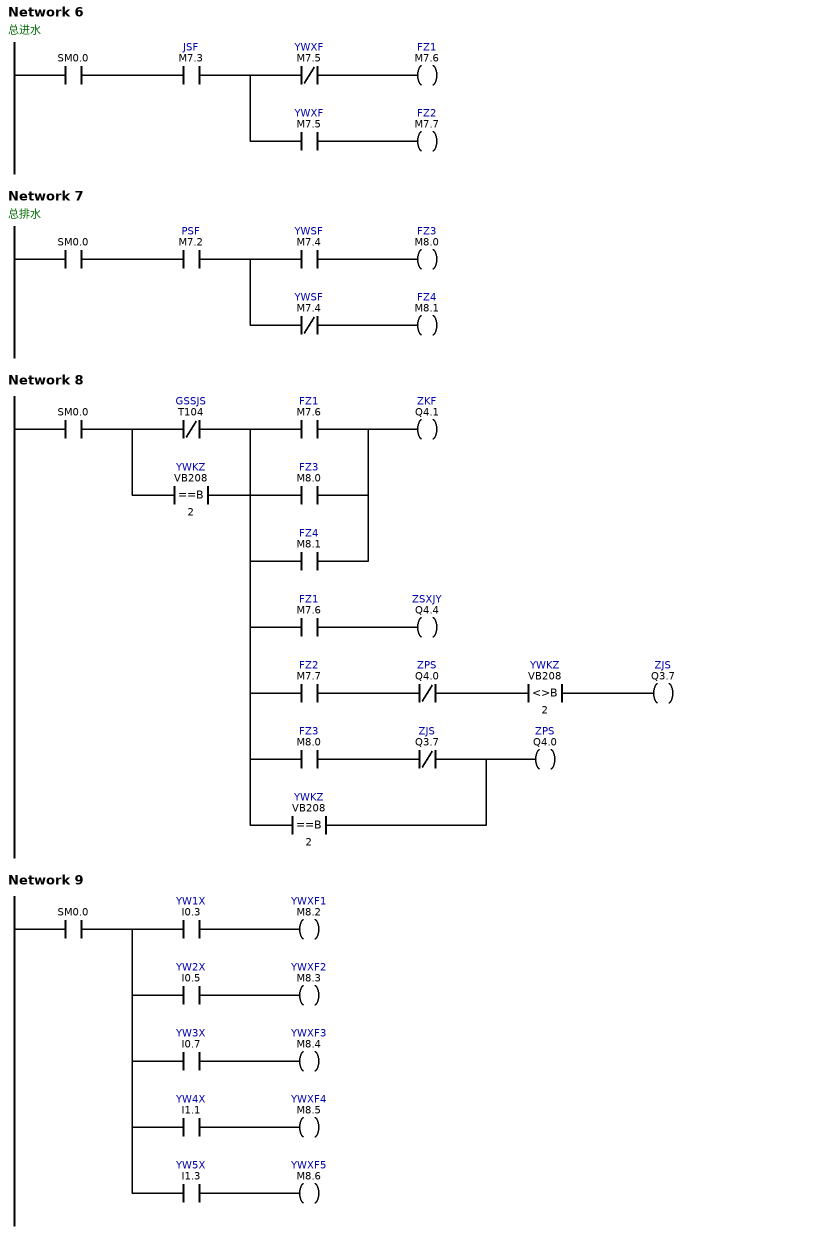
Network 6
// 总进水
LD     SM0.0
A      JSF:M7.3
LPS
AN     YWXF:M7.5
=      FZ1:M7.6
LPP
A      YWXF:M7.5
=      FZ2:M7.7
Network 7
// 总排水
LD     SM0.0
A      PSF:M7.2
LPS
A      YWSF:M7.4
=      FZ3:M8.0
LPP
AN     YWSF:M7.4
=      FZ4:M8.1
Network 8
LD     SM0.0
LDN    GSSJS:T104
OB=    YWKZ:VB208, 2
ALD
LPS
LD     FZ1:M7.6
O      FZ3:M8.0
O      FZ4:M8.1
ALD
=      ZKF:Q4.1
LRD
LPS
A      FZ1:M7.6
=      ZSXJY:Q4.4
LPP
A      FZ2:M7.7
AN     ZPS:Q4.0
AB<>   YWKZ:VB208, 2
=      ZJS:Q3.7
LPP
LD     FZ3:M8.0
AN     ZJS:Q3.7
OB=    YWKZ:VB208, 2
ALD
=      ZPS:Q4.0
Network 9
LD     SM0.0
LPS
A      YW1X:I0.3
=      YWXF1:M8.2
LRD
A      YW2X:I0.5
=      YWXF2:M8.3
LRD
A      YW3X:I0.7
=      YWXF3:M8.4
LRD
A      YW4X:I1.1
=      YWXF4:M8.5
LPP
A      YW5X:I1.3
=      YWXF5:M8.6
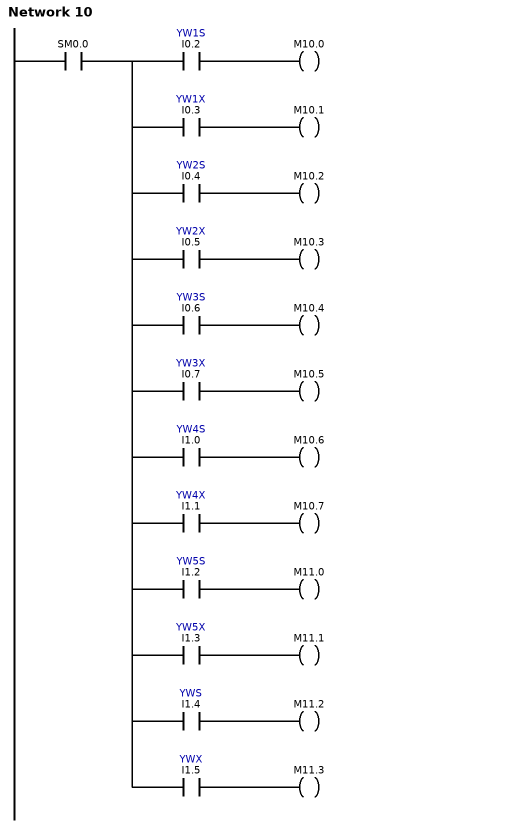
Network 10
LD     SM0.0
LPS
A      YW1S:I0.2
=      M10.0
LRD
A      YW1X:I0.3
=      M10.1
LRD
A      YW2S:I0.4
=      M10.2
LRD
A      YW2X:I0.5
=      M10.3
LRD
A      YW3S:I0.6
=      M10.4
LRD
A      YW3X:I0.7
=      M10.5
LRD
A      YW4S:I1.0
=      M10.6
LRD
A      YW4X:I1.1
=      M10.7
LRD
A      YW5S:I1.2
=      M11.0
LRD
A      YW5X:I1.3
=      M11.1
LRD
A      YWS:I1.4
=      M11.2
LPP
A      YWX:I1.5
=      M11.3
END_SUBROUTINE_BLOCK

SUBROUTINE_BLOCK HSC_初始化:SBR8
TITLE=子例行程序注释
BEGIN
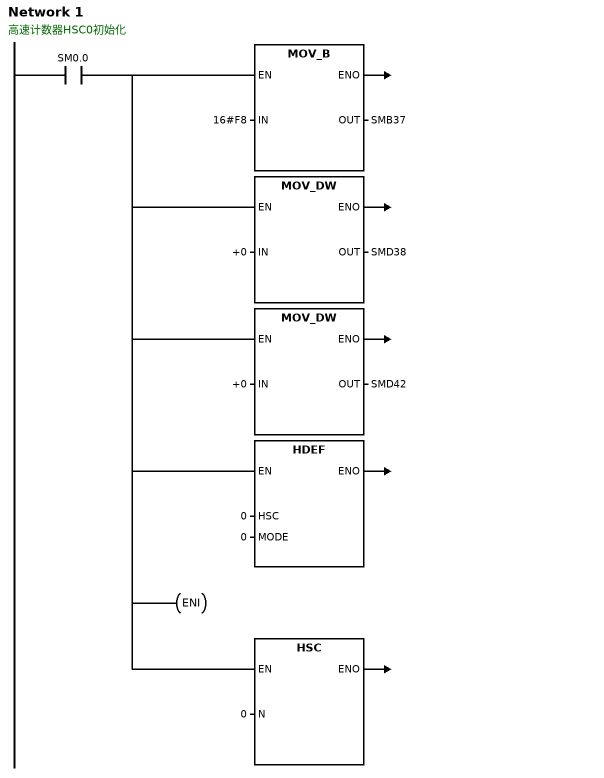
Network 1
// 高速计数器HSC0初始化
//设置控制位：向上计数；已启用；
//载入CV
//载入PV
LD     SM0.0
MOVB   16#F8, SMB37
MOVD   +0, SMD38
MOVD   +0, SMD42
HDEF   0, 0
ENI
HSC    0
Network 2 // 网络标题
// 网络注释
Network 12 // 网络标题
// 网络注释
Network 22 // 网络标题
// 网络注释
END_SUBROUTINE_BLOCK

SUBROUTINE_BLOCK 转速交变:SBR9
TITLE=采样延时
BEGIN
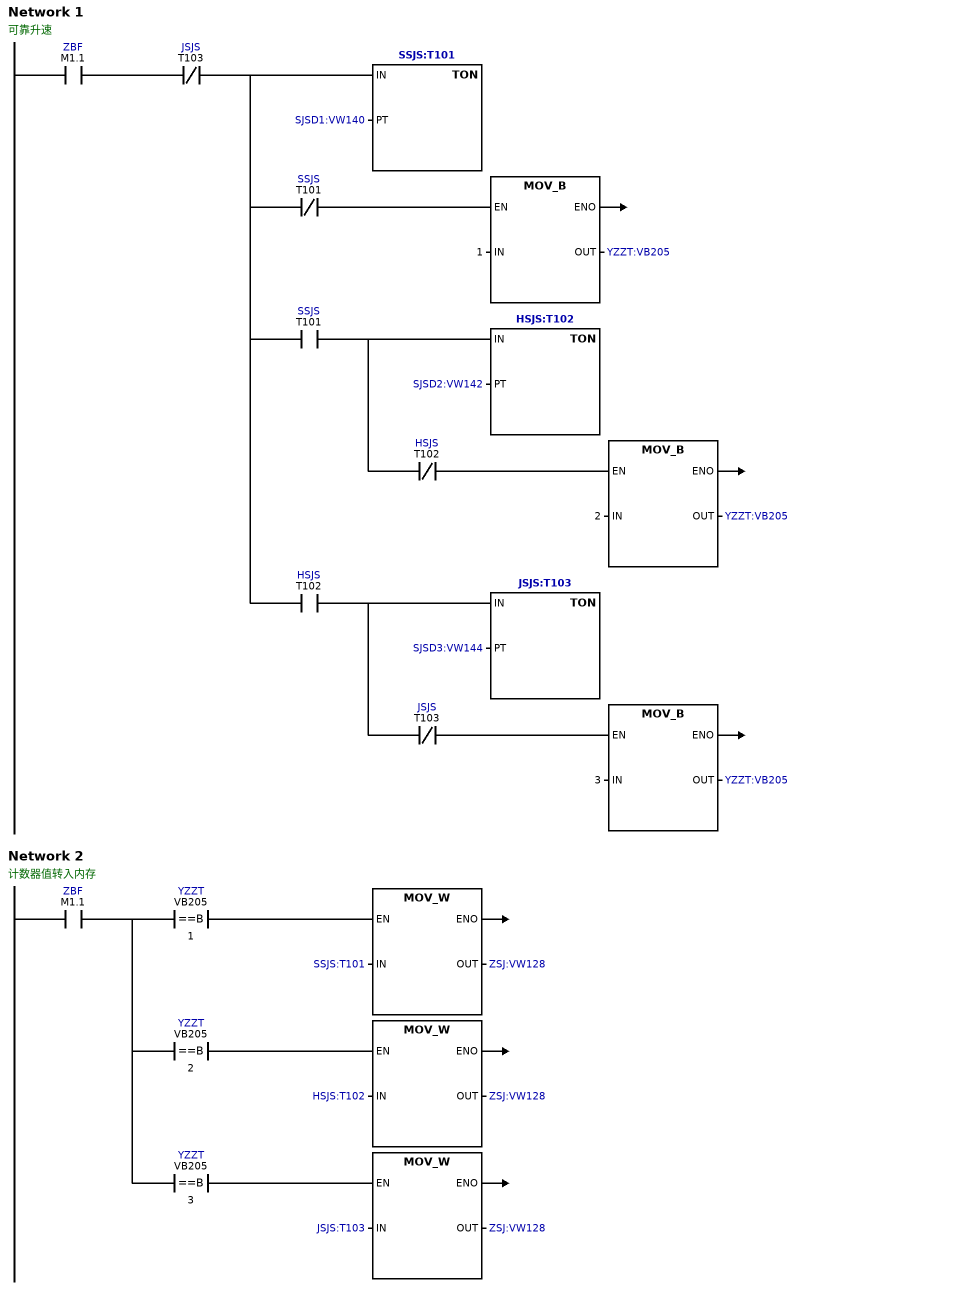
Network 1
// 可靠升速
LD     ZBF:M1.1
AN     JSJS:T103
LPS
TON    SSJS:T101, SJSD1:VW140
AN     SSJS:T101
MOVB   1, YZZT:VB205
LRD
A      SSJS:T101
TON    HSJS:T102, SJSD2:VW142
AN     HSJS:T102
MOVB   2, YZZT:VB205
LPP
A      HSJS:T102
TON    JSJS:T103, SJSD3:VW144
AN     JSJS:T103
MOVB   3, YZZT:VB205
Network 2
// 计数器值转入内存
LD     ZBF:M1.1
LPS
AB=    YZZT:VB205, 1
MOVW   SSJS:T101, ZSJ:VW128
LRD
AB=    YZZT:VB205, 2
MOVW   HSJS:T102, ZSJ:VW128
LPP
AB=    YZZT:VB205, 3
MOVW   JSJS:T103, ZSJ:VW128
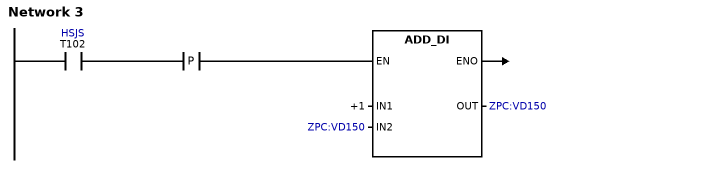
Network 3
LD     HSJS:T102
EU
+D     +1, ZPC:VD150
END_SUBROUTINE_BLOCK

SUBROUTINE_BLOCK 电阀控制:SBR10
TITLE=子例行程序注释
BEGIN
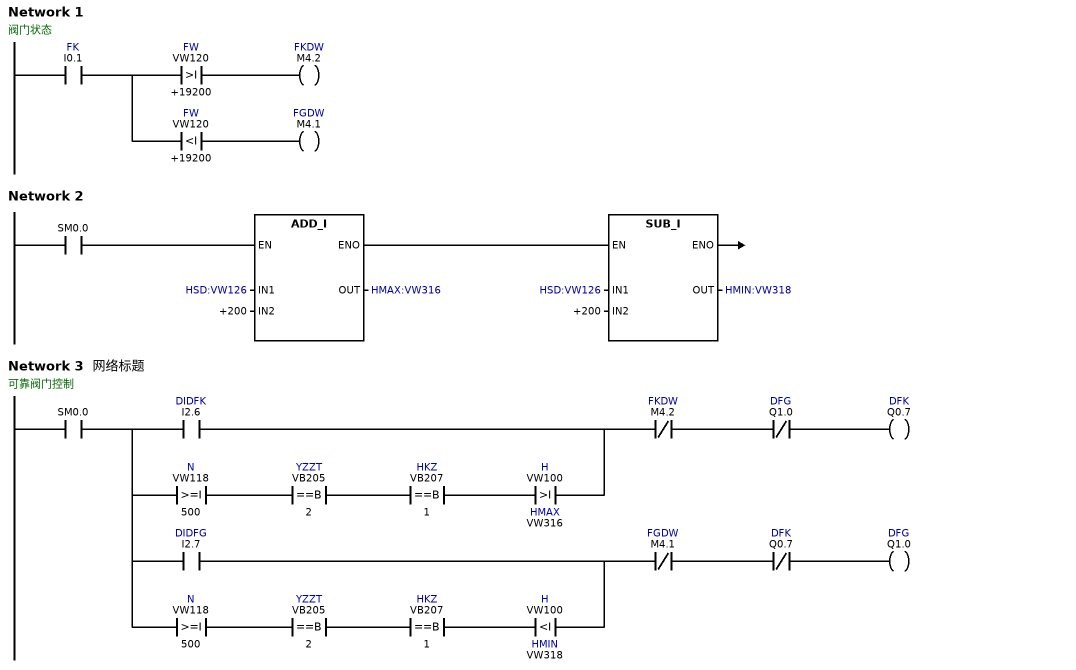
Network 1
// 阀门状态
LD     FK:I0.1
LPS
AW>    FW:VW120, +19200
=      FKDW:M4.2
LPP
AW<    FW:VW120, +19200
=      FGDW:M4.1
Network 2
LD     SM0.0
MOVW   HSD:VW126, HMAX:VW316
AENO
+I     +200, HMAX:VW316
AENO
MOVW   HSD:VW126, HMIN:VW318
-I     +200, HMIN:VW318
Network 3 // 网络标题
// 可靠阀门控制
LD     SM0.0
LPS
LD     DIDFK:I2.6
LDW>=  N:VW118, 500
AB=    YZZT:VB205, 2
AB=    HKZ:VB207, 1
AW>    H:VW100, HMAX:VW316
OLD
ALD
AN     FKDW:M4.2
AN     DFG:Q1.0
=      DFK:Q0.7
LPP
LD     DIDFG:I2.7
LDW>=  N:VW118, 500
AB=    YZZT:VB205, 2
AB=    HKZ:VB207, 1
AW<    H:VW100, HMIN:VW318
OLD
ALD
AN     FGDW:M4.1
AN     DFK:Q0.7
=      DFG:Q1.0
END_SUBROUTINE_BLOCK

SUBROUTINE_BLOCK 压力控制:SBR13
TITLE=子程序注释
BEGIN
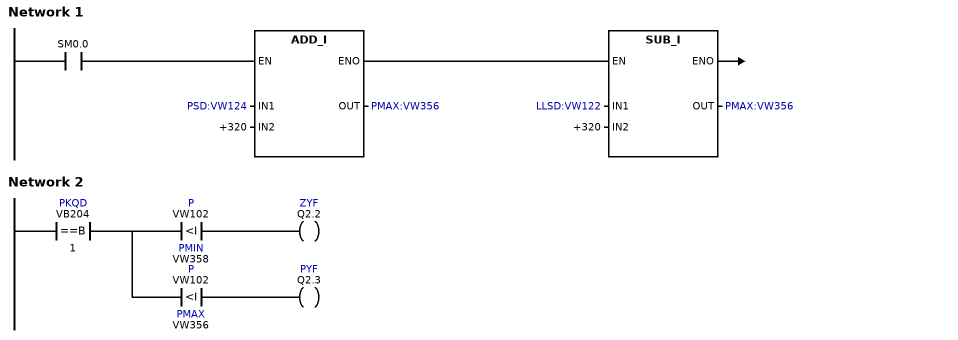
Network 1
LD     SM0.0
MOVW   PSD:VW124, PMAX:VW356
AENO
+I     +320, PMAX:VW356
AENO
MOVW   LLSD:VW122, PMAX:VW356
-I     +320, PMAX:VW356
Network 2
LDB=   PKQD:VB204, 1
LPS
AW<    P:VW102, PMIN:VW358
=      ZYF:Q2.2
LPP
AW<    P:VW102, PMAX:VW356
=      PYF:Q2.3
END_SUBROUTINE_BLOCK

INTERRUPT_BLOCK INT_1:INT1
TITLE=中断例行程序注释
BEGIN
